INTERFACE I_Device EXTENDS __SYSTEM.IQueryInterface

PROPERTY busy : BOOl
GET
END_GET
END_PROPERTY

PROPERTY done : BOOl
GET
END_GET
END_PROPERTY

PROPERTY error : BOOl
GET
END_GET
END_PROPERTY

PROPERTY id : DWORD
GET
END_GET
END_PROPERTY

PROPERTY ready : BOOl
GET
END_GET
END_PROPERTY

METHOD reset : BOOL
VAR_INPUT
END_VAR
END_METHOD

PROPERTY sid : STRING(255)
GET
END_GET
END_PROPERTY

END_INTERFACE

(* stored: Version 1.1.0.1, ProductVersion 3.1.4024.10
   Itf I_Device: Id {2fc5a503-fdad-4768-a08e-f93f94c2babe}
   Property busy: Id {b4eb8c30-02d8-47f0-bb8a-7a55e4b4fc0a}
   Get Get: Id {3241c714-7662-4c29-bfc8-17d565d8c38c}
   Property done: Id {cdb3fbf0-8d39-42e6-98f9-0edd27d42dde}
   Get Get: Id {abbb6683-c3de-4a90-ae46-f942ab099e08}
   Property error: Id {0f6e5059-0bc6-4c27-a25e-34282f0546b3}
   Get Get: Id {08004633-c587-4ea2-8c3a-b4bc760519dc}
   Property id: Id {b14a437d-9ce8-4776-9e9d-ed3e5979b12a}
   Get Get: Id {f9463c8b-2fbc-467e-a25e-5fd4cfe161c3}
   Property ready: Id {b5d6fcfd-8511-4477-a34e-7cbba0562119}
   Get Get: Id {00534eea-c00f-40b6-a599-6fa8e6c4ad94}
   Method reset: Id {286e3c18-0d10-4da5-b240-a9affe0a31c2}
   Property sid: Id {038e55bf-4b28-42cf-ba92-157227d63ae5}
   Get Get: Id {fb6b78ad-ba49-48a5-8915-b4c286f259ec} *)
